Omron Sysmac Studio project MODBUS_TCP_IP_SERVER_CONECT_HMI (Sysmac Studio 1.47.0.64008, StandardProject)

# Controller new_Controller_0: NX1P2-9024DT version 1.40
Task PrimaryTask (priority 4, period or condition 2000): Program0
Library OEN_Communication_V1_0_22 1.0.22 (contents left out)

VAR_GLOBAL
    NX1P2_OUT_0 : BOOL;  (* output_nx1p2; at BuiltInIO://cpu/#0/Output_Bit_00 *)
    NX1P2_OUT_1 : BOOL;  (* output_nx1p2; at BuiltInIO://cpu/#0/Output_Bit_01 *)
    NX1P2_OUT_2 : BOOL;  (* output_nx1p2; at BuiltInIO://cpu/#0/Output_Bit_02 *)
    NX1P2_OUT_3 : BOOL;  (* output_nx1p2; at BuiltInIO://cpu/#0/Output_Bit_03 *)
    NX1P2_OUT_4 : BOOL;  (* output_nx1p2; at BuiltInIO://cpu/#0/Output_Bit_04 *)
    NX1P2_OUT_5 : BOOL;  (* output_nx1p2; at BuiltInIO://cpu/#0/Output_Bit_05 *)
    NX1P2_OUT_6 : BOOL;  (* output_nx1p2; at BuiltInIO://cpu/#0/Output_Bit_06 *)
    NX1P2_OUT_7 : BOOL;  (* output_nx1p2; at BuiltInIO://cpu/#0/Output_Bit_07 *)
    NX1P2_OUT_8 : BOOL;  (* output_nx1p2; at BuiltInIO://cpu/#0/Output_Bit_08 *)
    NX1P2_OUT_9 : BOOL;  (* output_nx1p2; at BuiltInIO://cpu/#0/Output_Bit_09 *)
    NX1P2_IN_3 : BOOL;  (* IN_NX1P2_9024DT; at BuiltInIO://cpu/#0/Input_Bit_03 *)
    NX1P2_IN_4 : BOOL;  (* IN_NX1P2_9024DT; at BuiltInIO://cpu/#0/Input_Bit_04 *)
    NX1P2_IN_5 : BOOL;  (* IN_NX1P2_9024DT; at BuiltInIO://cpu/#0/Input_Bit_05 *)
    NX1P2_IN_6 : BOOL;  (* IN_NX1P2_9024DT; at BuiltInIO://cpu/#0/Input_Bit_06 *)
    NX1P2_IN_1 : BOOL;  (* IN_NX1P2_9024DT; at BuiltInIO://cpu/#0/Input_Bit_01 *)
    NX1P2_IN_2 : BOOL;  (* IN_NX1P2_9024DT; at BuiltInIO://cpu/#0/Input_Bit_02 *)
    NX1P2_IN_0 : BOOL;  (* IN_NX1P2_9024DT; at BuiltInIO://cpu/#0/Input_Bit_00 *)
    NX1P2_IN_7 : BOOL;  (* IN_NX1P2_9024DT; at BuiltInIO://cpu/#0/Input_Bit_07 *)
    NX1P2_IN_8 : BOOL;  (* IN_NX1P2_9024DT; at BuiltInIO://cpu/#0/Input_Bit_08 *)
    NX1P2_IN_9 : BOOL;  (* IN_NX1P2_9024DT; at BuiltInIO://cpu/#0/Input_Bit_09 *)
    NX1P2_IN_10 : BOOL;  (* IN_NX1P2_9024DT; at BuiltInIO://cpu/#0/Input_Bit_10 *)
    NX1P2_IN_11 : BOOL;  (* IN_NX1P2_9024DT; at BuiltInIO://cpu/#0/Input_Bit_11 *)
    NX1P2_IN_12 : BOOL;  (* IN_NX1P2_9024DT; at BuiltInIO://cpu/#0/Input_Bit_12 *)
    NX1P2_IN_13 : BOOL;  (* IN_NX1P2_9024DT; at BuiltInIO://cpu/#0/Input_Bit_13 *)
END_VAR

PROGRAM Program0
VAR
    TCP_SERVER_CONNECT : BOOL;
    FB_TCP_SERVER : OEN\Modbus\ModbusTCP_Server;
    DATA_ACCESS_LIST : ARRAY[0..10] OF OEN\Modbus\sModbusAccess := [4((RegisterType := Coil, AccessType := R, AddressArea := (StartAddress := 0, Count := 0))), (RegisterType := Coil, AccessType := RW, AddressArea := (StartAddress := 0, Count := 0)), 6((RegisterType := Coil, AccessType := R, AddressArea := (StartAddress := 0, Count := 0)))];
    MODBUS_COIL : ARRAY[0..10] OF BOOL;
    DISCRETE_INPUT : ARRAY[0..10] OF BOOL;
    MODBUS_DISCRETE_INPUT : ARRAY[0..10] OF BOOL;
    INPUT_RES : ARRAY[0..10] OF WORD;
    HOLDING_REGISTER : ARRAY[0..10] OF WORD;
    TRANSFER_RES : ARRAY[0..11] OF WORD;
    T0_TCP : TON;
    T1_TCP : TON;
END_VAR
VAR_EXTERNAL
    NX1P2_OUT_0 : BOOL;
    NX1P2_OUT_1 : BOOL;
END_VAR

(* Section Section0: ladder, written here as Structured Text *)

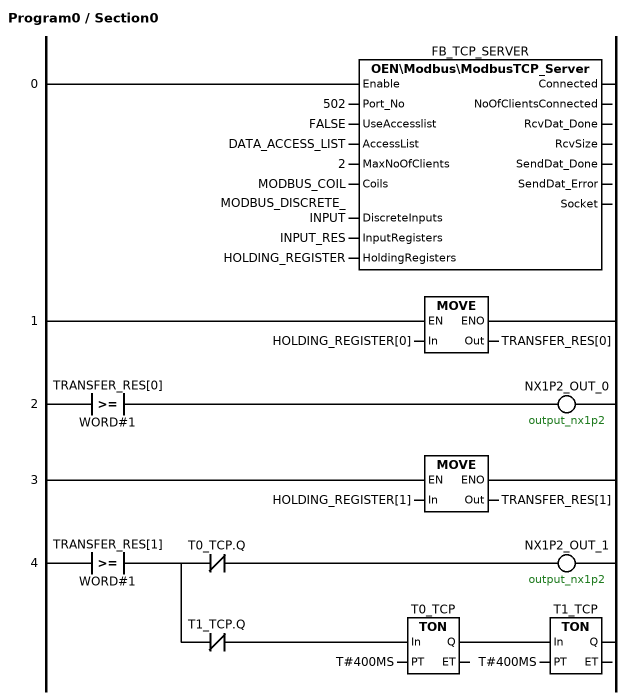
(* Rung 0 *)
FB_TCP_SERVER(Enable := TRUE, Port_No := 502, UseAccesslist := FALSE, AccessList := DATA_ACCESS_LIST, MaxNoOfClients := 2, Coils := MODBUS_COIL, DiscreteInputs := MODBUS_DISCRETE_INPUT, InputRegisters := INPUT_RES, HoldingRegisters := HOLDING_REGISTER);
(* Rung 1 *)
TRANSFER_RES[0] := HOLDING_REGISTER[0];
(* Rung 2 *)
NX1P2_OUT_0 := TRANSFER_RES[0] >= WORD#1;
(* Rung 3 *)
TRANSFER_RES[1] := HOLDING_REGISTER[1];
(* Rung 4 *)
NX1P2_OUT_1 := (TRANSFER_RES[1] >= WORD#1) AND NOT T0_TCP.Q;
T0_TCP(In := (TRANSFER_RES[1] >= WORD#1) AND NOT T1_TCP.Q, PT := T#400MS);
T1_TCP(In := T0_TCP.Q, PT := T#400MS);
END_PROGRAM